// TwinCAT 3 PLC project Maschine
// ProgramVersion: 3.1.4024.0
// libraries:
//   Tc2_Standard, * (Beckhoff Automation GmbH)
//   Tc2_System, * (Beckhoff Automation GmbH)
//   Tc3_Module, * (Beckhoff Automation GmbH)
// project tree:
//   / PlcTask.TcTTO
//   POUs/ FB_TestMaschinentuer.TcPOU, MAIN.TcPOU
// (motion and I/O tree: see PLC project sps)
// real-time tasks:
//   TASK PlcTask: cycle T#10ms, priority 20, ADS port 350
//   TASK PlcTask1: cycle T#10ms, priority 21, ADS port 351
// variable links:

CONFIGURATION Maschine
    RESOURCE PLC ON TwinCAT3
        TASK PlcTask(INTERVAL := T#10ms, PRIORITY := 21);
        PROGRAM MAIN WITH PlcTask : MAIN;
    END_RESOURCE
END_CONFIGURATION

// ---- POUs/MAIN.TcPOU
PROGRAM MAIN
VAR
	bDoorC AT%Q* : BOOL;
	bDoorO AT%Q* : BOOL;
	bVentil AT%I* : BOOL;
	
	fbTestMaschinentuer : FB_TestMaschinentuer;
END_VAR


fbTestMaschinentuer(bVentil:= bVentil ,
 					bDoorC=> bDoorC , 
					bDoorO=> bDoorO);

END_PROGRAM

// ---- POUs/FB_TestMaschinentuer.TcPOU
FUNCTION_BLOCK FB_TestMaschinentuer
VAR_INPUT
	bVentil : BOOL;
END_VAR
VAR_OUTPUT
	bDoorC : BOOL := TRUE;
	bDoorO : BOOL;
END_VAR
VAR
	RTrig : R_Trig;
	FTrig : F_Trig;
	fbTon1 : Ton;
	fbTon2 : Ton;
END_VAR

FTrig(CLK:= bVentil, Q=> );
RTrig(CLK:= bVentil, Q=> );
fbTon1(PT:= T#1S);
fbTon2(PT:= T#1S);

IF Ftrig.Q THEN
	fbTon1.IN := TRUE;
	bDoorC := FALSE;
END_IF
	IF fbTon1.Q THEN
		bDoorO := TRUE;
		fbTon1.IN := FALSE;
	END_IF



IF RTrig.Q THEN
	fbTon2.In := TRUE;
	bDoorO := FALSE;
END_IF
	IF fbTon2.Q THEN
		bDoorC := TRUE;
		fbTon2.IN := FALSE;
	END_IF

END_FUNCTION_BLOCK
